PROGRAM MAIN
VAR
	stDataHMI : ST_HMIManager;
END_VAR

END_PROGRAM

(* stored: Version 1.1.0.1
   POU MAIN: Id {488fd77b-6a8e-4774-9619-09a4fd5cfcbc}, SpecialFunc None *)
